// HW status for control cabinet alarms and rotation drive
TYPE ST_HW_STATUS_DEV :
STRUCT	
	bEStopOK:BOOL;                       // s2: ch1: emergency stop ok                 Verify: OK   
	bRF02_MainDriveThermalFilterOK:BOOL; // s2: ch2: rf01 termal braking filter OK..   Verify: Q to Markus: Maybe this should be rf02?
	bTA01_TA02_24VSupplyOK:BOOL;         // s2: ch3: ta01 and ta02 24V power supply OK Verify: OK  
	bFC11_Fuse24VOK:BOOL;                // s2: ch4: fc11 24V fuse OK                   Verify: OK
	bFA01_FA02_OvervoltageOK:BOOL;       // s2: ch5: fa01 and fa02 overvoltage protection OK
	bFC01_FuseMainRotationOK:BOOL;       // s2: ch6: fc01 fuse target wheel motor OK
	bFC06_FC07_FuseICSOutletsOK:BOOL;    // s2: ch7: fc06 and fc07 ICS outlets fuse OK
	bFC51_FC52_FC53_FuseUPSOK:BOOL;      // s2: ch8: fc51, fc52 and fc53 UPS fuses OK (something wrong)
	
	// Bridge terminal EL6695
	bBeamOff:BOOL; 
	
END_STRUCT
END_TYPE

(* stored: Version 1.1.0.1, ProductVersion 3.1.4024.6
   DUT ST_HW_STATUS_DEV: Id {4425b300-01a1-4265-9988-b6ed7e8d4e9d} *)
